SUBAPPLICATION Blocker (* Subapplication Type *)
  (* Standard: 61499-2 *)
  (* Version 1.0, 2018-09-13, az *)
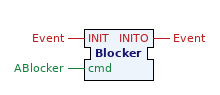
  EVENT_INPUT
    INIT;
  END_EVENT
  EVENT_OUTPUT
    INITO;
  END_EVENT
  SOCKETS
    cmd : ABlocker;
  END_SOCKETS
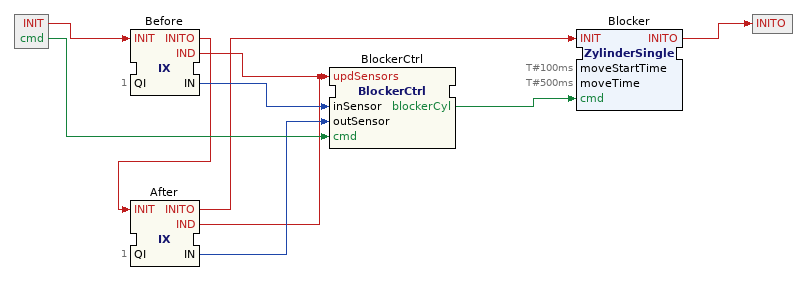
  FBS
    After : IX(QI := 1);
    Before : IX(QI := 1);
    BlockerCtrl : BlockerCtrl;
  END_FBS
  SUBAPPS
    Blocker : ZylinderSingle(moveStartTime := T#100ms, moveTime := T#500ms);
  END_SUBAPPS
  EVENT_CONNECTIONS
    Before.INITO TO After.INIT;
    INIT TO Before.INIT;
    After.INITO TO Blocker.INIT;
    Blocker.INITO TO INITO;
    Before.IND TO BlockerCtrl.updSensors;
    After.IND TO BlockerCtrl.updSensors;
  END_CONNECTIONS
  DATA_CONNECTIONS
    Before.IN TO BlockerCtrl.inSensor;
    After.IN TO BlockerCtrl.outSensor;
  END_CONNECTIONS
  ADAPTER_CONNECTIONS
    cmd TO BlockerCtrl.cmd;
    BlockerCtrl.blockerCyl TO Blocker.cmd;
  END_CONNECTIONS
END_SUBAPPLICATION
